TYPE CameraRecipe :
STRUCT
	ExposureTime : UDINT;
	RulerLines : UDINT;
END_STRUCT
END_TYPE

(* stored: Version 1.1.0.1
   DUT CameraRecipe: Id {9af1d9a7-afb1-42aa-9e4b-57e0a91690ee} *)
